{attribute addProperty BoxType "EL6851-0000-0017"}
{attribute addProperty Id "ChannelAT %Q*ARRAY[0 ..63] OF USINT512640"}
{attribute addProperty CRC "1632717686"}
{attribute addProperty SizeInBites "512"}
{attribute addProperty SizeInBytes "64"}
TYPE DMX_Channel_59324749 :
STRUCT
	{attribute addProperty Name "Channel"}
	Channel AT %Q* : ARRAY[0 ..63] OF USINT;
END_STRUCT
END_TYPE

(* stored: Version 1.2.0.0, ProductVersion 3.1.4024.9
   DUT DMX_Channel_59324749: Id {d0d78c0c-ed4e-4898-92ce-d2eff9d581ad} *)
